TYPE OP120_Recipe :
STRUCT
	OP120_Bowl_Feeder_Freq:LREAL;
	OP120_Robo_Prog_No:INT;
	OP120_Camera_Prog_No:INT;
	
END_STRUCT
END_TYPE

(* stored: Version 1.1.0.1, ProductVersion 3.1.4024.11
   DUT OP120_Recipe: Id {3b98861b-5d3d-4db9-a06a-48a02550de65} *)
